{attribute addProperty BoxType "EL5002-0000-0016"}
{attribute addProperty Id "SSI_Inputs_ChannelAT %I*ARRAY[0..1] OF SSI_Inputs_Channel_F7D238D196120WcStateAT %I*WcState_98A4DF7520.250InfoDataAT %I*InfoData_BC63D37F80100"}
{attribute addProperty CRC "4210564609"}
{attribute addProperty SizeInBites "178"}
{attribute addProperty SizeInBytes "22.25"}
TYPE EL5002_82283068 :
STRUCT
	{attribute addProperty Name "SSI_Inputs_Channel"}
	SSI_Inputs_Channel : ARRAY[0..1] OF SSI_Inputs_Channel_F7D238D1;
	{attribute addProperty Name "WcState"}
	WcState : WcState_98A4DF75;
	{attribute addProperty Name "InfoData"}
	InfoData : InfoData_BC63D37F;
END_STRUCT
END_TYPE

(* stored: Version 1.2.0.0, ProductVersion 3.1.4024.9
   DUT EL5002_82283068: Id {29682185-d92b-468a-89a1-c564f609eaf5} *)
